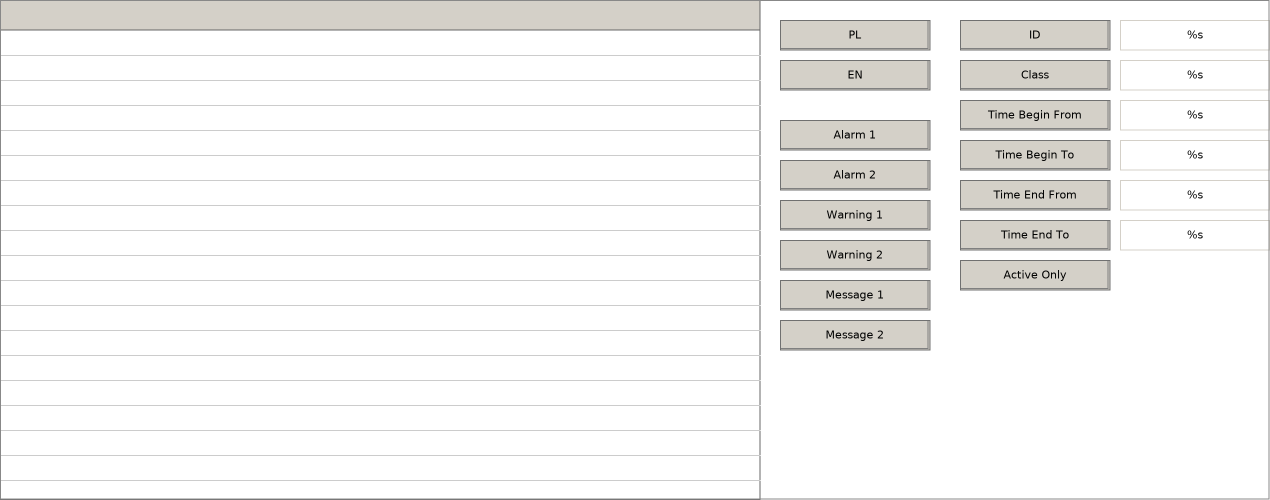
VISUALIZATION VISU_EventsHistoricalSimple  // 1270x500
    Group (780,120 150x230)
        Button (0,0 150x30), "Alarm 1", colour toggle: GVL_EHS.arrEventDefinition[1].bActive
            toggle GVL_EHS.arrEventDefinition[1].bActive
        Button (0,40 150x30), "Alarm 2", colour toggle: GVL_EHS.arrEventDefinition[2].bActive
            toggle GVL_EHS.arrEventDefinition[2].bActive
        Button (0,80 150x30), "Warning 1", colour toggle: GVL_EHS.arrEventDefinition[31].bActive
            toggle GVL_EHS.arrEventDefinition[31].bActive
        Button (0,120 150x30), "Warning 2", colour toggle: GVL_EHS.arrEventDefinition[32].bActive
            toggle GVL_EHS.arrEventDefinition[32].bActive
        Button (0,160 150x30), "Message 1", colour toggle: GVL_EHS.arrEventDefinition[41].bActive
            toggle GVL_EHS.arrEventDefinition[41].bActive
        Button (0,200 150x30), "Message 2", colour toggle: GVL_EHS.arrEventDefinition[42].bActive
            toggle GVL_EHS.arrEventDefinition[42].bActive
    Group (780,20 150x70)
        Button (0,0 150x30), "PL"
            OnMouseDown: execute { GVL_EHS.dwLanguageId := 1045; }
        Button (0,40 150x30), "EN"
            OnMouseDown: execute { GVL_EHS.dwLanguageId := 1033; }
    Table (0,0 760x500), data array: GVL_EHS.arrEventVisu
        p3854506369: GVL_EHS.arrEventVisu[INDEX].dwID
        p1892666644: GVL_EHS.arrEventVisu[INDEX].dwParam
        p338671338: GVL_EHS.arrEventVisu[INDEX].wsMessage
        p2170511999: GVL_EHS.arrEventVisu[INDEX].dtDateBegin
        p3723444502: GVL_EHS.arrEventVisu[INDEX].dtDateEnd
        p511219082: Class
        p2237128397: Date Begin
        p505689113: Date End
        p3312258591: GVL_EHS.arrEventVisu[INDEX].dwClass
        Columns.Column.[2].Template: GVL_EHS.arrEventVisu[INDEX].dwColor
    Group (960,20 310x270)
        Button (0,0 150x30), "ID", colour toggle: P_EventsVisuHS.bFilterID
            toggle P_EventsVisuHS.bFilterID
        Button (0,40 150x30), "Class", colour toggle: P_EventsVisuHS.bFilterClass
            toggle P_EventsVisuHS.bFilterClass
        Button (0,80 150x30), "Time Begin From", colour toggle: P_EventsVisuHS.bFilterBeginTimeFrom
            toggle P_EventsVisuHS.bFilterBeginTimeFrom
        Button (0,120 150x30), "Time Begin To", colour toggle: P_EventsVisuHS.bFilterBeginTimeTo
            toggle P_EventsVisuHS.bFilterBeginTimeTo
        Button (0,160 150x30), "Time End From", colour toggle: P_EventsVisuHS.bFilterEndTimeFrom
            toggle P_EventsVisuHS.bFilterEndTimeFrom
        Button (0,200 150x30), "Time End To", colour toggle: P_EventsVisuHS.bFilterEndTimeTo
            toggle P_EventsVisuHS.bFilterEndTimeTo
        Button (0,240 150x30), "Active Only", colour toggle: P_EventsVisuHS.bFilterActiveOnly
            toggle P_EventsVisuHS.bFilterActiveOnly
        Textfield (160,0 150x30), "%s", text variable: P_EventsVisuHS.dwFilterID
            OnMouseDown: write the text variable via VisuDialogs.Numpad
        Textfield (160,40 150x30), "%s", text variable: P_EventsVisuHS.dwFilterClass
            OnMouseDown: write the text variable via VisuDialogs.Numpad
        Textfield (160,80 150x30), "%s", text variable: P_EventsVisuHS.dtFilterBeginTimeFrom
            OnMouseDown: write the text variable via Edit
        Textfield (160,120 150x30), "%s", text variable: P_EventsVisuHS.dtFilterBeginTimeTo
            OnMouseDown: write the text variable via Edit
        Textfield (160,160 150x30), "%s", text variable: P_EventsVisuHS.dtFilterEndTimeFrom
            OnMouseDown: write the text variable via Edit
        Textfield (160,200 150x30), "%s", text variable: P_EventsVisuHS.dtFilterEndTimeTo
            OnMouseDown: write the text variable via Edit
END_VISUALIZATION

(* stored: Version 1.1.0.1, ProductVersion 3.1.4024.3
   Visu VISU_EventsHistoricalSimple: Id {0e80b0d0-6086-4047-90d2-da838d9cb3f3} *)
